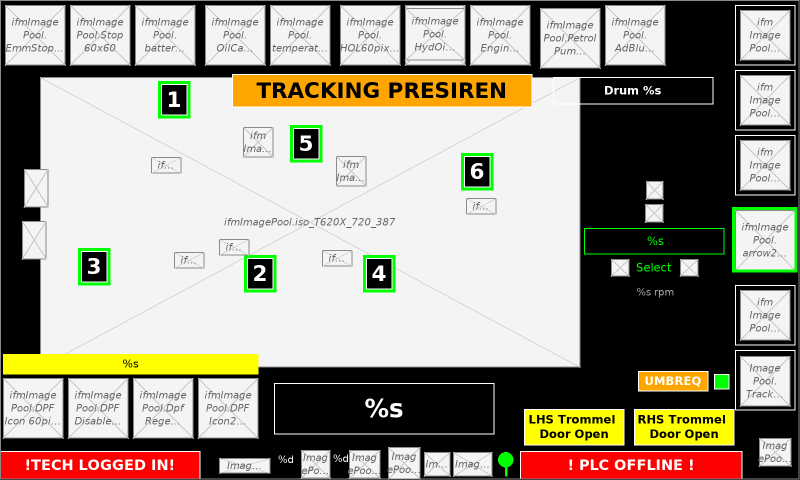
VISUALIZATION Visualization_Main_1  // 800x480
    Frame (0,0 800x480)
        shows Visualization_Main_Status_Common()
    Frame (0,0 800x480)
        shows Visualization_Template()
    Frame (0,0 800x480)
        shows Visualization_Main_Status_Common()
        shows Visualization_Main_Status_Radial()
    Image (740,10 50x50), invisible if: AutoManSelButtons.AutoStartShow=0, image: ifmImagePool.start50pixel
    Image (740,75 50x50), invisible if: AutoManSelButtons.AutoStopShow=0, image: ifmImagePool.Stop Button50pixel
    RoundedRectangle (735,5 60x60)
    RoundedRectangle (735,70 60x60)
    RoundedRectangle (735,135 60x60)
    RoundedRectangle (735,285 60x60)
    RoundedRectangle (735,350 60x60)
    Image (740,140 50x50), image: ifmImagePool.Maintenance50pixel
    RoundedRectangle (735,350 60x60)
    Image (740,290 50x50), image: ifmImagePool.speedometer50pixel
    Image (735,210 60x60), image: ifmImagePool.arrow2_60pixel
    RoundedRectangle (732,207 65x65), invisible if: AutoManSelButtons.Mimic_Halo_RPM_Up_Down=0
        p3450524324: GVL_Viz.SelColor_DWORD
    Image (740,356 50x50), image: ImagePool.Track_50_50
    Rectangle (714,374 15x15), invisible if: GVL_Machine.TrackingModeAllow=0
    RoundedRectangle (524,409 100x36), "LHS Trommel Door Open", invisible if: Machine_IO.Inputs.LHS_TROMMELDOORSW.Dig
    RoundedRectangle (634,409 100x36), "RHS Trommel Door Open", invisible if: Machine_IO.Inputs.RHS_TROMMELDOORSW.Dig
    RoundedRectangle (553,77 160x27), "Drum %s", text variable: GVL_Machine.DrumPressMsg
    RoundedRectangle (638,371 70x20), "UMBREQ", invisible if: Machine_IO.Inputs.UMBTRACKREQ.Dig=0
END_VISUALIZATION

// Device/Application/App_Common/Vizualisations/Main/Visualization_Engine_1
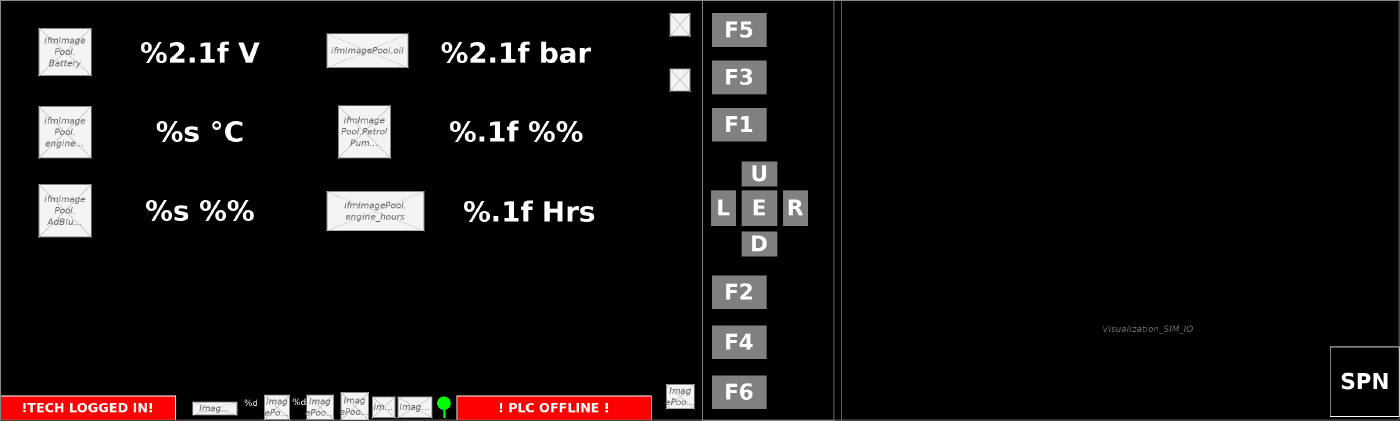
VISUALIZATION Visualization_Engine_1  // 1595x480
    Frame (0,0 800x480)
        shows Visualization_Template()
    Image (385,120 60x60), image: ifmImagePool.Petrol Pump60pixel
    Rectangle (100,20 256x81), "%2.1f V", text variable: GVL_Engine.EngineVoltage
    RoundedRectangle (1515,395 80x80), "SPN"
    Rectangle (460,20 256x81), "%2.1f bar", text variable: GVL_Engine.OilPress_bar/100
    Rectangle (100,110 256x81), "%s °C", text variable: GVL_Engine.CoolantTemperature_degC
    Rectangle (100,200 256x81), "%s %%", text variable: GVL_Engine.Def_TankLevelPercent
    Rectangle (490,201 226x81), "%.1f Hrs", text variable: GVL_Engine.EngineHrs
    Image (385,120 60x60), image: ifmImagePool.Petrol Pump60pixel
    Image (385,120 60x60), invisible if: GVL_Alarms.LowFuelAlarm=0, image: ifmImagePool.Petrol PumpRed60pixel
    Rectangle (460,110 256x81), "%.1f %%", text variable: Machine_IO.Inputs.FUELLEVEL_PERCENT.ScaledReal
    Image (44,210 60x60), image: ifmImagePool.AdBlue Icon On Black60pixel
    Image (372,38 93x39), image: ifmImagePool.oil
    Image (44,121 60x59), image: ifmImagePool.engine_temp
    Image (44,32 60x54), image: ifmImagePool.Battery
    Image (372,218 111x45), image: ifmImagePool.engine_hours
    Image (763,15 23x26), invisible if: Nav.Footer_ShowNavLeft=0, image: ImagePool.Page_nav_left
    Image (763,78 23x26), invisible if: Nav.Footer_ShowNavRight=0, image: ImagePool.Page_nav_right
END_VISUALIZATION

// Device/Application/App_Common/Vizualisations/Main/Visualization_Engine_2
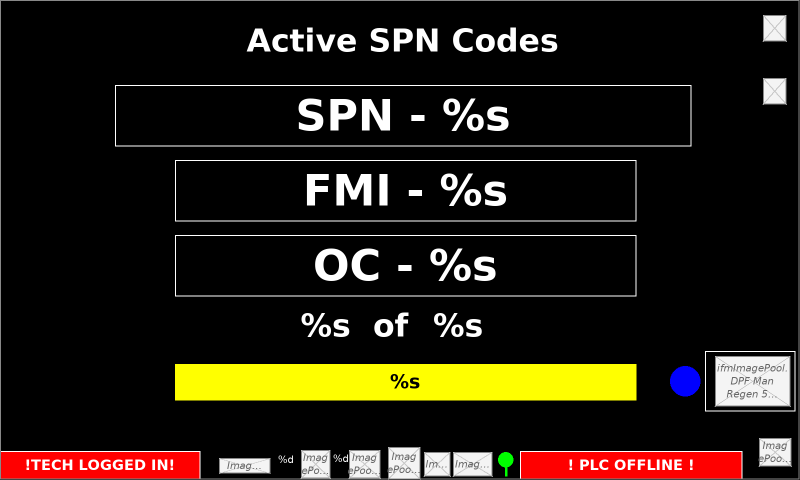
VISUALIZATION Visualization_Engine_2  // 800x480
    Frame (0,0 800x480)
        shows Visualization_Template()
    Rectangle (115,15 576x51), "Active SPN Codes"
    Rectangle (115,85 576x61), "SPN - %s", text variable: GVL_Engine.DM1_Index_SPN
    Rectangle (175,160 461x61), "FMI - %s", text variable: GVL_Engine.DM1_Index_FMI
    Rectangle (175,235 461x61), "OC - %s", text variable: GVL_Engine.DM1_Index_OC
    Rectangle (175,300 236x51), "%s of", text variable: GVL_Engine.DM1_Index
    Rectangle (430,300 206x51), "%s", text variable: GVL_Engine.QtyOf_SPN_Codes
    Image (715,356 75x50), image: ifmImagePool.DPF Man Regen 50 pixelhigh
    Ellipse (670,366 30x30), invisible if: GVL_Engine.ElevateRpmAllowed=FALSE
    RoundedRectangle (705,351 90x60)
    Image (763,15 23x26), invisible if: Nav.Footer_ShowNavLeft=0, image: ImagePool.Page_nav_left
    Image (763,78 23x26), invisible if: Nav.Footer_ShowNavRight=0, image: ImagePool.Page_nav_right
    RoundedRectangle (175,364 461x36), "%s", text variable: GVL_Engine.DPF_Regen_Status_String
END_VISUALIZATION

// Device/Application/App_Common/Vizualisations/Main/Visualization_Settings_2
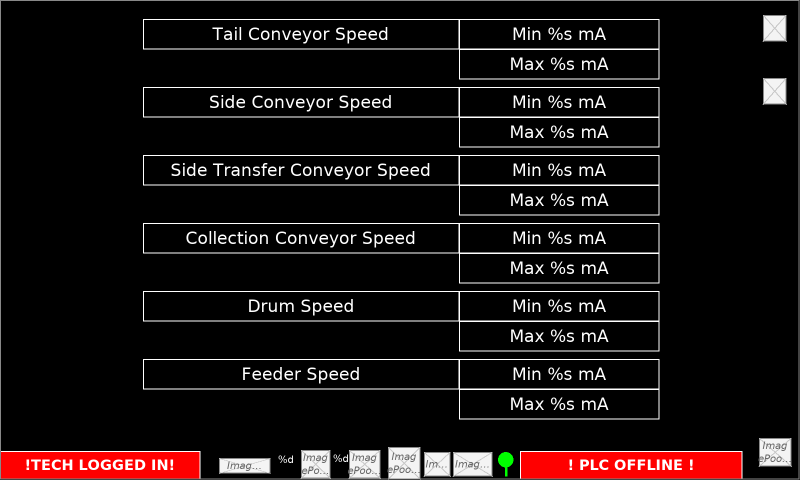
VISUALIZATION Visualization_Settings_2  // 800x480
    Frame (0,0 800x480)
        shows Visualization_Template()
    Rectangle (459,19 200x30), "Min %s mA", text variable: GVL_Persistant.App_Settings.TailConvSpd_Min_mA
        OnMouseClick: write the text variable via VisuDialogs_Template.Numpad, min 0, max GVL_Persistant.App_Settings.TailConvSpd_Max_mA, title "Tail Conveyor Speed Min"
    Rectangle (143,19 316x30), "Tail Conveyor Speed"
    Rectangle (459,49 200x30), "Max %s mA", text variable: GVL_Persistant.App_Settings.TailConvSpd_Max_mA
        OnMouseClick: write the text variable via VisuDialogs_Template.Numpad, min GVL_Persistant.App_Settings.TailConvSpd_Min_mA, max GVL_Persistant.App_Settings.Valve_mA_Max, title "Tail Conveyor Speed Max"
    Rectangle (459,87 200x30), "Min %s mA", text variable: GVL_Persistant.App_Settings.SideConvSpd_Min_mA
        OnMouseClick: write the text variable via VisuDialogs_Template.Numpad, min 0, max GVL_Persistant.App_Settings.SideConvSpd_Max_mA, title "Side Conveyor Speed Min"
    Rectangle (143,87 316x30), "Side Conveyor Speed"
    Rectangle (459,117 200x30), "Max %s mA", text variable: GVL_Persistant.App_Settings.SideConvSpd_Max_mA
        OnMouseClick: write the text variable via VisuDialogs_Template.Numpad, min GVL_Persistant.App_Settings.SideConvSpd_Min_mA, max GVL_Persistant.App_Settings.Valve_mA_Max, title "Side Conveyor Speed Max"
    Rectangle (459,155 200x30), "Min %s mA", text variable: GVL_Persistant.App_Settings.SideTransferConvSpd_Min_mA
        OnMouseClick: write the text variable via VisuDialogs_Template.Numpad, min 0, max GVL_Persistant.App_Settings.SideTransferConvSpd_Max_mA, title "Side Transfer Conveyor Speed Min"
    Rectangle (143,155 316x30), "Side Transfer Conveyor Speed"
    Rectangle (459,185 200x30), "Max %s mA", text variable: GVL_Persistant.App_Settings.SideTransferConvSpd_Max_mA
        OnMouseClick: write the text variable via VisuDialogs_Template.Numpad, min GVL_Persistant.App_Settings.SideTransferConvSpd_Min_mA, max GVL_Persistant.App_Settings.Valve_mA_Max, title "Side Transfer Conveyor Speed Max"
    Rectangle (459,223 200x30), "Min %s mA", text variable: GVL_Persistant.App_Settings.CollectConvSpd_Min_mA
        OnMouseClick: write the text variable via VisuDialogs_Template.Numpad, min 0, max GVL_Persistant.App_Settings.CollectConvSpd_Max_mA, title "Collection Conveyor Speed Min"
    Rectangle (143,223 316x30), "Collection Conveyor Speed"
    Rectangle (459,253 200x30), "Max %s mA", text variable: GVL_Persistant.App_Settings.CollectConvSpd_Max_mA
        OnMouseClick: write the text variable via VisuDialogs_Template.Numpad, min GVL_Persistant.App_Settings.CollectConvSpd_Min_mA, max GVL_Persistant.App_Settings.Valve_mA_Max, title "Collection Conveyor Speed Max"
    Rectangle (459,291 200x30), "Min %s mA", text variable: GVL_Persistant.App_Settings.DrumSpd_Min_mA
        OnMouseClick: write the text variable via VisuDialogs_Template.Numpad, min 0, max GVL_Persistant.App_Settings.DrumSpd_Max_mA, title "Drum Speed Min"
    Rectangle (143,291 316x30), "Drum Speed"
    Rectangle (459,321 200x30), "Max %s mA", text variable: GVL_Persistant.App_Settings.DrumSpd_Max_mA
        OnMouseClick: write the text variable via VisuDialogs_Template.Numpad, min GVL_Persistant.App_Settings.DrumSpd_Min_mA, max GVL_Persistant.App_Settings.Valve_mA_Max, title "Drum Speed Max"
    Rectangle (459,359 200x30), "Min %s mA", text variable: GVL_Persistant.App_Settings.FeederSpd_Min_mA
        OnMouseClick: write the text variable via VisuDialogs_Template.Numpad, min 0, max GVL_Persistant.App_Settings.FeederSpd_Max_mA, title "Feeder Speed Min"
    Rectangle (143,359 316x30), "Feeder Speed"
    Rectangle (459,389 200x30), "Max %s mA", text variable: GVL_Persistant.App_Settings.FeederSpd_Max_mA
        OnMouseClick: write the text variable via VisuDialogs_Template.Numpad, min GVL_Persistant.App_Settings.FeederSpd_Min_mA, max GVL_Persistant.App_Settings.Valve_mA_Max, title "Feeder Speed Max"
    Image (763,15 23x26), invisible if: Nav.Footer_ShowNavLeft=0, image: ImagePool.Page_nav_left
    Image (763,78 23x26), invisible if: Nav.Footer_ShowNavRight=0, image: ImagePool.Page_nav_right
END_VISUALIZATION

// Device/Application/App_Common/Vizualisations/Main/Layout/Visualization_Main_Status_Common
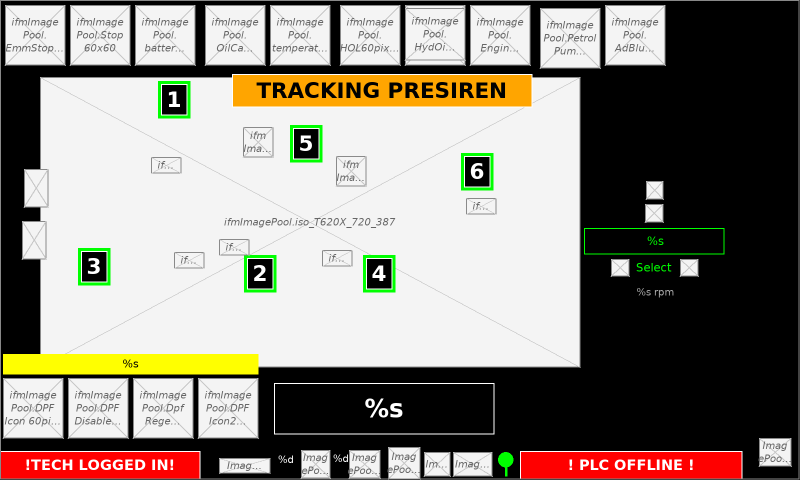
VISUALIZATION Visualization_Main_Status_Common  // 800x480
    Frame (0,0 800x480)
        shows Visualization_Template()
    Frame (0,0 800x480), frame switch variable: TO_INT(GVL_APP.MachineModelRadial)
        shows Visualization_Main_Status_Standard()
        shows Visualization_Main_Status_Radial()
    Image (135,5 60x60), invisible if: GVL_Machine.ChargeLamp=FALSE, image: ifmImagePool.batteryREDonBlack60pixel
    Image (205,5 60x60), invisible if: GVL_Engine.EngineLowOilPressAlarm=FALSE, image: ifmImagePool.OilCanREDonBlack60pixel
    Image (270,5 60x60), invisible if: GVL_Engine.EngineHiTempAlarm=FALSE, image: ifmImagePool.temperatureREDonBlack60pixel
    Image (340,5 60x60), invisible if: GVL_Alarms.LowHydOilAlarm=FALSE, image: ifmImagePool.HOL60pixel
    Image (405,5 60x60), invisible if: GVL_Alarms.HydTempAlarm=FALSE, image: ifmImagePool.HydOilTemp60pixel
    Image (5,5 60x60), invisible if: Safety_Common.ESTOP_HEALHTY_COMMON=0, image: ifmImagePool.EmmStop60pixel
    Image (198,378 60x60), invisible if: GVL_Engine.MILamp=FALSE, image: ifmImagePool.DPF Icon2_60pixel
    Image (133,378 60x60), invisible if: GVL_Engine.DPF_RegenActive=FALSE, image: ifmImagePool.Dpf Regen Active60pixel
    Image (68,378 60x60), invisible if: GVL_Engine.DPF_Regen_Inhibited=FALSE, image: ifmImagePool.DPF Disabled Lamp60pixel
    Image (3,378 60x60), invisible if: GVL_Engine.DPF_Lamp=FALSE, image: ifmImagePool.DPF Icon 60pixel
    Image (70,5 60x60), invisible if: GVL_Machine.UmbMachineShutdown=FALSE, image: ifmImagePool.Stop 60x60
    Image (605,5 60x60), invisible if: GVL_Engine.Def_LowLevLamp=FALSE, image: ifmImagePool.AdBlue Icon On Black60pixel
    Image (470,5 60x60), invisible if: GVL_Engine.EngineWarningLamp=FALSE, image: ifmImagePool.Engine IconAmber60pixel
    Image (470,5 60x60), invisible if: GVL_Engine.DisplayEngineStopLamp=FALSE, image: ifmImagePool.Engine IconRed60pixel
    Image (540,8 60x60), invisible if: PLC_Alarms.Fuel_Symbol_Visible=0, image: ifmImagePool.Petrol PumpRed60pixel
    RoundedRectangle (274,383 220x51), "%s", text variable: GVL_Engine.EngineRpmPerctangeString
    Image (405,8 60x52), invisible if: GVL_Alarms.DrumHighPress_Alarm=0, image: ifmImagePool.HydOil Warning 60 pixel
    RoundedRectangle (232,74 300x33), "TRACKING MODE", invisible if: GVL_Machine.TrackingMode=0
    RoundedRectangle (232,74 300x33), "TRACKING PRESIREN", invisible if: GVL_Machine.TrackPreSiren_Flash=0
    RoundedRectangle (3,354 255x20), "%s", text variable: GVL_Engine.DPF_Regen_Status_String, invisible if: GVL_Engine.DPF_Regen_Status=0
    RoundedRectangle (584,228 140x26), "%s", text variable: AutoManSelButtons.Selected_String, invisible if: LEN(AutoManSelButtons.Selected_String)=0
    Image (646,181 17x18), invisible if: AutoManSelButtons.NavUpShow=0, image: ImagePool.Nav_Up_17_18
    Image (646,204 17x18), invisible if: AutoManSelButtons.NavDownShow=0, image: ImagePool.Nav_Down_17_18
    Image (645,204 18x18), invisible if: AutoManSelButtons.NavCirleShow=0, image: ImagePool.NavCircle_18_18
    Image (611,259 18x17), invisible if: AutoManSelButtons.NavLeftShow=0, image: ImagePool.Nav_Left_17_18
    Image (680,259 18x17), invisible if: AutoManSelButtons.NavRightShow=0, image: ImagePool.Nav_Right_17_18
    RoundedRectangle (629,259 50x17), "Select", text variable: AutoManSelButtons.Selected_String, invisible if: AutoManSelButtons.NavSelectShow=0
    RoundedRectangle (584,279 140x26), "%s rpm", text variable: GVL_Engine.RequestedRPM, invisible if: LEN(AutoManSelButtons.Selected_String)=0
END_VISUALIZATION

// Device/Application/App_Common/Vizualisations/Main/Visualization_Settings_4
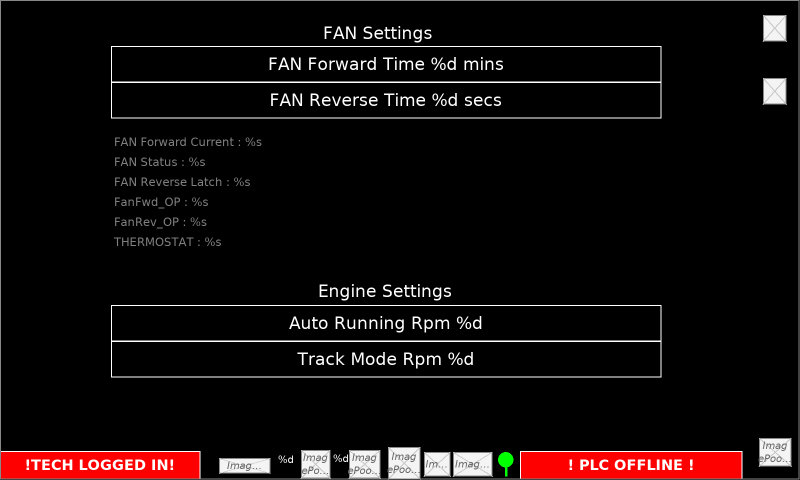
VISUALIZATION Visualization_Settings_4  // 800x480
    Frame (0,0 800x480)
        shows Visualization_Template()
        OnMouseClick: write the text variable via Default, min 0, max 3600, title "Drum Cutout"
    Rectangle (111,46 550x36), "FAN Forward Time %d mins", text variable: GVL_Persistant.App_Settings.Fan_FwdTime_mins
        OnMouseClick: write the text variable via VisuDialogs_Template.Numpad, min 5, max 60, title "FAN Foward Time (mins)"
    Rectangle (155,5 446x56), "FAN Settings"
    Image (763,15 23x26), invisible if: Nav.Footer_ShowNavLeft=0, image: ImagePool.Page_nav_left
    Image (763,78 23x26), invisible if: Nav.Footer_ShowNavRight=0, image: ImagePool.Page_nav_right
    Rectangle (111,82 550x36), "FAN Reverse Time %d secs", text variable: GVL_Persistant.App_Settings.Fan_RevTime_secs
        OnMouseClick: write the text variable via VisuDialogs_Template.Numpad, min 30, max 1200, title "FAN Reverse Time"
    Rectangle (111,132 550x20), "FAN Forward Current : %s", text variable: PLC_FanCtrl.Current_Forward_Time_STR
    Rectangle (111,152 550x20), "FAN Status : %s", text variable: PLC_FanCtrl.STATUS_STRING
    Rectangle (111,172 550x20), "FAN Reverse Latch : %s", text variable: GVL_Persistant.App_Run_Vars.Fan_Reverse_Latch
    Rectangle (111,192 550x20), "FanFwd_OP : %s", text variable: TO_BOOL(Machine_IO.Outputs.FanFwd_OP.Dig)
    Rectangle (111,212 550x20), "FanRev_OP : %s", text variable: TO_BOOL(Machine_IO.Outputs.FanRev_OP.Dig)
    Rectangle (111,232 550x20), "THERMOSTAT : %s", text variable: PLC_FanCtrl.THERMOSTAT
    Rectangle (111,305 550x36), "Auto Running Rpm %d", text variable: GVL_Persistant.App_Settings.AutoRunningRpm
        OnMouseClick: write the text variable via VisuDialogs_Template.Numpad, min GVL_Persistant.App_Settings.AutoRunningRpmMin, max GVL_Persistant.App_Settings.AutoRunningRpmMax, title "Auto Running Rpm"
    Rectangle (162,263 446x56), "Engine Settings"
    Rectangle (111,341 550x36), "Track Mode Rpm %d", text variable: GVL_Persistant.App_Settings.TrackModeRpm
        OnMouseClick: write the text variable via VisuDialogs_Template.Numpad, min GVL_Persistant.App_Settings.TrackModeRpmMin, max GVL_Persistant.App_Settings.TrackModeRpmMax, title "Auto Running Rpm"
END_VISUALIZATION

// /Visualization
VISUALIZATION Visualization  // 1024x768
END_VISUALIZATION

// /Visualization_1
VISUALIZATION Visualization_1  // 1024x768
END_VISUALIZATION

// Device/Application/App_Common/Vizualisations/DIAG_IO/Visualization_DIAG_IO_AUX
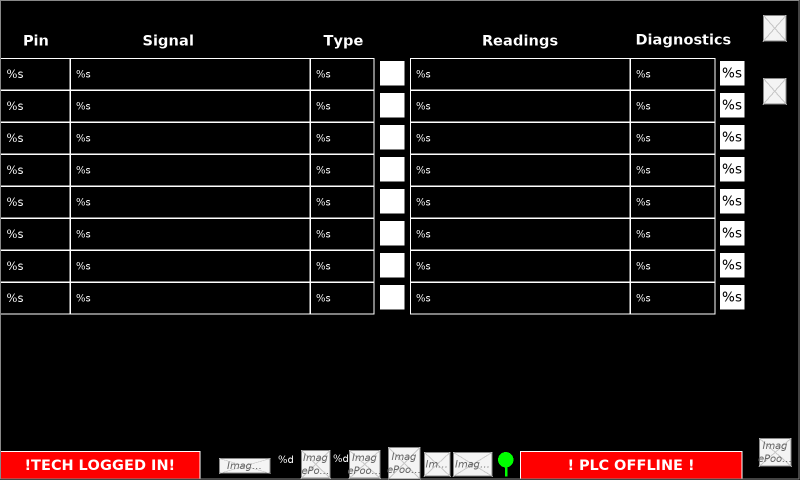
VISUALIZATION Visualization_DIAG_IO_AUX  // 800x480
    Frame (0,0 800x480)
        shows Visualization_Template()
    Image (763,15 23x26), invisible if: Nav.Footer_ShowNavLeft=0, image: ImagePool.Page_nav_left
    Image (763,78 23x26), invisible if: Nav.Footer_ShowNavRight=0, image: ImagePool.Page_nav_right
    Frame (0,25 750x420)
        shows Visualization_CR0403_Op()
END_VISUALIZATION

// Device/Application/App_Common/Vizualisations/DIAG_IO/CR0403/Output_IFM_PLC_CR0403
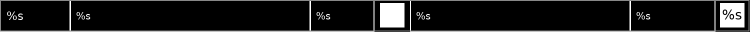
VISUALIZATION Output_IFM_PLC_CR0403  // 750x32
VAR_IN_OUT
	Output: CR0403_Output_Display;
END_VAR
VAR
END_VAR
    Textfield (70,0 240x32), "%s", text variable: Output.oSignalNameStr
    Textfield (0,0 70x32), "%s", text variable: Output.oPinDetailsStr
    Rectangle (380,3 24x24), invisible if: NOT Output.oShowDigRect, colour variable: Output.oDigRectColour
        p3450524324: Output.oDigRectColour
    Textfield (310,0 64x32), "%s", text variable: Output.oTypeStr
    Rectangle (720,3 24x24), "%s", text variable: Output.oForceText, invisible if: NOT HMI_IO.Outputs_EnableAutoMan, input disabled if: NOT HMI_IO.Outputs_EnableAutoMan OR GVL_System.HMI_OP_FORCE_DISABLE, colour variable: Output.oForceColour
        p3450524324: Output.oForceColour
        OnMouseClick:  Dialog=Output_Force, Parameters={flags: , pOutputState: Output.OpREF.OUTPUT_STATE_DATA}, Selected={1: , 0: }, OpenModal=True, OpenCentered=True
    Textfield (630,0 85x32), "%s", text variable: Output.oDiagStr
        p55702900: Output.oMainStringColour
    Textfield (410,0 220x32), "%s", text variable: Output.oMainString
        p55702900: Output.oMainStringColour
END_VISUALIZATION

// Device/Application/App_Common/Vizualisations/DIAG_IO/CR0403/Visualization_CR0403_Op
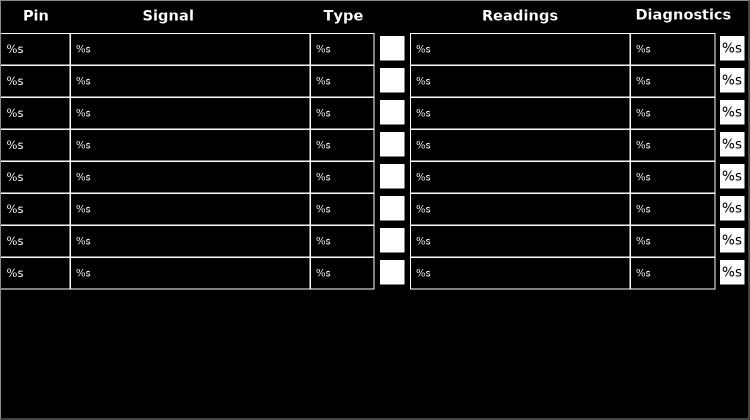
VISUALIZATION Visualization_CR0403_Op  // 750x420
    Frame (0,0 800x32)
        shows Output_IFM_PLC_CRXXXX_TITLE()
    Frame (0,33 750x32)
        shows Output_IFM_PLC_CR0403(Output := HMI_IO.AUX.OP0)
    Frame (0,65 750x32)
        shows Output_IFM_PLC_CR0403(Output := HMI_IO.AUX.OP1)
    Frame (0,97 750x32)
        shows Output_IFM_PLC_CR0403(Output := HMI_IO.AUX.OP2)
    Frame (0,129 750x32)
        shows Output_IFM_PLC_CR0403(Output := HMI_IO.AUX.OP3)
    Frame (0,161 750x32)
        shows Output_IFM_PLC_CR0403(Output := HMI_IO.AUX.OP4)
    Frame (0,193 750x32)
        shows Output_IFM_PLC_CR0403(Output := HMI_IO.AUX.OP5)
    Frame (0,225 750x32)
        shows Output_IFM_PLC_CR0403(Output := HMI_IO.AUX.OP6)
    Frame (0,257 750x32)
        shows Output_IFM_PLC_CR0403(Output := HMI_IO.AUX.OP7)
END_VISUALIZATION

// Device/Application/App_Common/Vizualisations/Main/Layout/Visualization_Main_Status_Radial
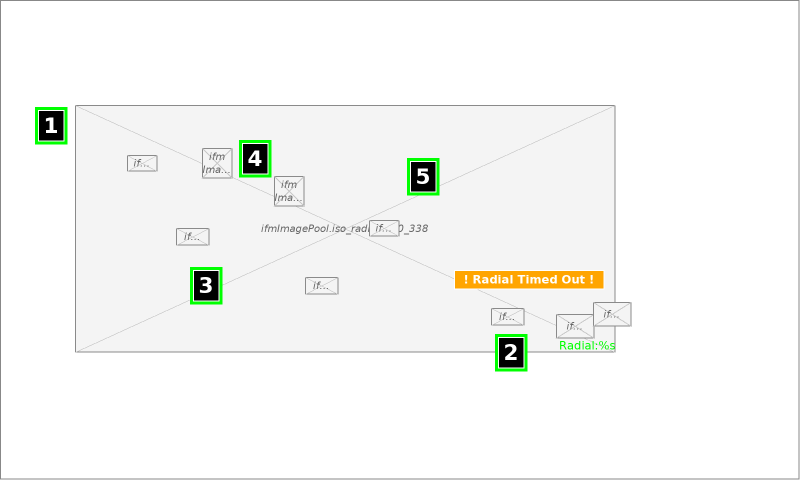
VISUALIZATION Visualization_Main_Status_Radial  // 800x480
    Image (75,105 540x247), image: ifmImagePool.iso_radial_720_338
    Image (369,220 30x16), angle 200, invisible if: Page_Ctrl.Radial_Feeder.Invisible, image: ifmImagePool.Right Arrow Simple 30 pixel wide
        p3560616238: Page_Ctrl.Radial_Feeder.OutX
        p2738717112: Page_Ctrl.Radial_Feeder.OutY
    RoundedRectangle (38,110 26x31), "1", colour variable: AutoManSelButtons.Icon_1_Fill_Colour
    RoundedRectangle (498,337 26x31), "2", colour variable: AutoManSelButtons.Icon_2_Fill_Colour
    RoundedRectangle (410,161 26x31), "5", colour variable: AutoManSelButtons.Icon_5_Fill_Colour
    RoundedRectangle (193,270 26x31), "3", colour variable: AutoManSelButtons.Icon_3_Fill_Colour
    RoundedRectangle (242,143 26x31), "4", colour variable: AutoManSelButtons.Icon_4_Fill_Colour
    Image (274,176 30x30), invisible if: Page_Ctrl.DrumArrow.Invisible, image: ifmImagePool.Rotating Arrow30pixel
        p2858320360: Page_Ctrl.DrumArrow.Out+90
    RoundedRectangle (35,107 32x37), invisible if: AutoManSelButtons.Mimic_Halo_1=0
        p3450524324: GVL_Viz.SelColor_DWORD
    RoundedRectangle (495,334 32x37), invisible if: AutoManSelButtons.Mimic_Halo_2=0
        p3450524324: GVL_Viz.SelColor_DWORD
    RoundedRectangle (239,140 32x37), invisible if: AutoManSelButtons.Mimic_Halo_4=0
        p3450524324: GVL_Viz.SelColor_DWORD
    RoundedRectangle (407,158 32x37), invisible if: AutoManSelButtons.Mimic_Halo_5=0
        p3450524324: GVL_Viz.SelColor_DWORD
    Image (202,148 30x30), invisible if: Page_Ctrl.DrumArrow.Invisible, image: ifmImagePool.Rotating Arrow30pixel
        p2858320360: Page_Ctrl.DrumArrow.Out
    Image (176,228 33x17), angle 22, invisible if: Page_Ctrl.Radial_CollectionArrow_Flat.Invisible, image: ifmImagePool.Right Arrow Simple 30 pixel wide
        p3560616238: Page_Ctrl.Radial_CollectionArrow_Flat.OutX
        p2738717112: Page_Ctrl.Radial_CollectionArrow_Flat.OutY
    Image (491,308 33x17), angle -12, invisible if: Page_Ctrl.Radial_StockpileArrow.Invisible, image: ifmImagePool.Right Arrow Simple 30 pixel wide
        p3560616238: Page_Ctrl.Radial_StockpileArrow.OutX
        p2738717112: Page_Ctrl.Radial_StockpileArrow.OutY
    Image (127,155 30x16), angle 229, invisible if: Page_Ctrl.Radial_TailConveyor.Invisible, image: ifmImagePool.Right Arrow Simple 30 pixel wide
        p3560616238: Page_Ctrl.Radial_TailConveyor.OutX
        p2738717112: Page_Ctrl.Radial_TailConveyor.OutY
    Image (305,277 33x17), angle -1, invisible if: Page_Ctrl.Radial_CollectionArrow_Flat.Invisible, image: ifmImagePool.Right Arrow Simple 30 pixel wide
        p3560616238: Page_Ctrl.Radial_CollectionArrow_Ramp.OutX
        p2738717112: Page_Ctrl.Radial_CollectionArrow_Ramp.OutY
    RoundedRectangle (190,267 32x37), invisible if: AutoManSelButtons.Mimic_Halo_3=0
        p3450524324: GVL_Viz.SelColor_DWORD
    RoundedRectangle (454,270 150x19), "! Radial Timed Out !", invisible if: GVL_APP.RadialTimeOutFlag=0
    Image (556,314 38x24), invisible if: Machine_IO.Outputs.SideConvRaise_RadialLeft_OP.Dig=0, image: ifmImagePool.radial_right
    Image (593,302 38x24), invisible if: Machine_IO.Outputs.SideConvLower_RadialRight_OP.Dig=0, image: ifmImagePool.radial_left
    RoundedRectangle (556,336 150x19), "Radial:%s", text variable: PLC_RadialMode.STATUS_STRING
END_VISUALIZATION

// Device/Application/App_Common/Vizualisations/Main/Layout/Visualization_Main_Status_Standard
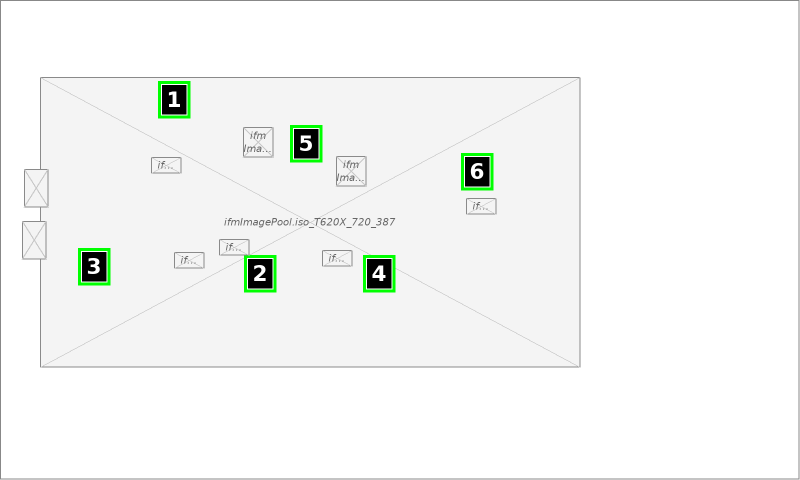
VISUALIZATION Visualization_Main_Status_Standard  // 800x480
    Image (40,77 540x290), image: ifmImagePool.iso_T620X_720_387
    Image (466,198 30x16), angle 198, invisible if: Page_Ctrl.Standard_FeederArrow.Invisible, image: ifmImagePool.Right Arrow Simple 30 pixel wide
        p3560616238: Page_Ctrl.Standard_FeederArrow.OutX
        p2738717112: Page_Ctrl.Standard_FeederArrow.OutY
    RoundedRectangle (161,84 26x31), "1", colour variable: AutoManSelButtons.Icon_1_Fill_Colour
    RoundedRectangle (81,251 26x31), "3", colour variable: AutoManSelButtons.Icon_3_Fill_Colour
    RoundedRectangle (464,156 26x31), "6", colour variable: AutoManSelButtons.Icon_6_Fill_Colour
    RoundedRectangle (293,128 26x31), "5", colour variable: AutoManSelButtons.Icon_5_Fill_Colour
    RoundedRectangle (247,258 26x31), "2", colour variable: AutoManSelButtons.Icon_2_Fill_Colour
    RoundedRectangle (366,258 26x31), "4", colour variable: AutoManSelButtons.Icon_4_Fill_Colour
    Image (322,250 30x16), angle 198, invisible if: Page_Ctrl.Standard_CollectionArrow.Invisible, image: ifmImagePool.Right Arrow Simple 30 pixel wide
        p3560616238: Page_Ctrl.Standard_CollectionArrow.OutX
        p2738717112: Page_Ctrl.Standard_CollectionArrow.OutY
    Image (243,127 30x30), invisible if: Page_Ctrl.DrumArrow.Invisible, image: ifmImagePool.Rotating Arrow30pixel
        p2858320360: Page_Ctrl.DrumArrow.Out
    RoundedRectangle (158,81 32x37), invisible if: AutoManSelButtons.Mimic_Halo_1=0
        p3450524324: GVL_Viz.SelColor_DWORD
    RoundedRectangle (244,255 32x37), invisible if: AutoManSelButtons.Mimic_Halo_2=0
        p3450524324: GVL_Viz.SelColor_DWORD
    RoundedRectangle (78,248 32x37), invisible if: AutoManSelButtons.Mimic_Halo_3=0
        p3450524324: GVL_Viz.SelColor_DWORD
    RoundedRectangle (363,255 32x37), invisible if: AutoManSelButtons.Mimic_Halo_4=0
        p3450524324: GVL_Viz.SelColor_DWORD
    RoundedRectangle (290,125 32x37), invisible if: AutoManSelButtons.Mimic_Halo_5=0
        p3450524324: GVL_Viz.SelColor_DWORD
    RoundedRectangle (461,153 32x37), invisible if: AutoManSelButtons.Mimic_Halo_6=0
        p3450524324: GVL_Viz.SelColor_DWORD
    Image (336,156 30x30), invisible if: Page_Ctrl.DrumArrow.Invisible, image: ifmImagePool.Rotating Arrow30pixel
        p2858320360: Page_Ctrl.DrumArrow.Out+90
    Image (174,252 30x16), angle 198, invisible if: Page_Ctrl.Standard_SideConvArrow.Invisible, image: ifmImagePool.Right Arrow Simple 30 pixel wide
        p3560616238: Page_Ctrl.Standard_SideConvArrow.OutX
        p2738717112: Page_Ctrl.Standard_SideConvArrow.OutY
    Image (219,239 30x16), angle 161, invisible if: Page_Ctrl.Standard_SideTransferArrow.Invisible, image: ifmImagePool.Right Arrow Simple 30 pixel wide
        p3560616238: Page_Ctrl.Standard_SideTransferArrow.OutX
        p2738717112: Page_Ctrl.Standard_SideTransferArrow.OutY
    Image (151,157 30x16), angle 224, invisible if: Page_Ctrl.Standard_TailConvArrow.Invisible, image: ifmImagePool.Right Arrow Simple 30 pixel wide
        p3560616238: Page_Ctrl.Standard_TailConvArrow.OutX
        p2738717112: Page_Ctrl.Standard_TailConvArrow.OutY
    Image (24,169 24x38), invisible if: Machine_IO.Outputs.SideConvRaise_RadialLeft_OP.Dig=0, image: ifmImagePool.side_conv_up
    Image (22,221 24x38), invisible if: Machine_IO.Outputs.SideConvLower_RadialRight_OP.Dig=0, image: ifmImagePool.side_conv_down
END_VISUALIZATION

// Device/Application/App_Common/Vizualisations/Main/Visualization_Settings_3
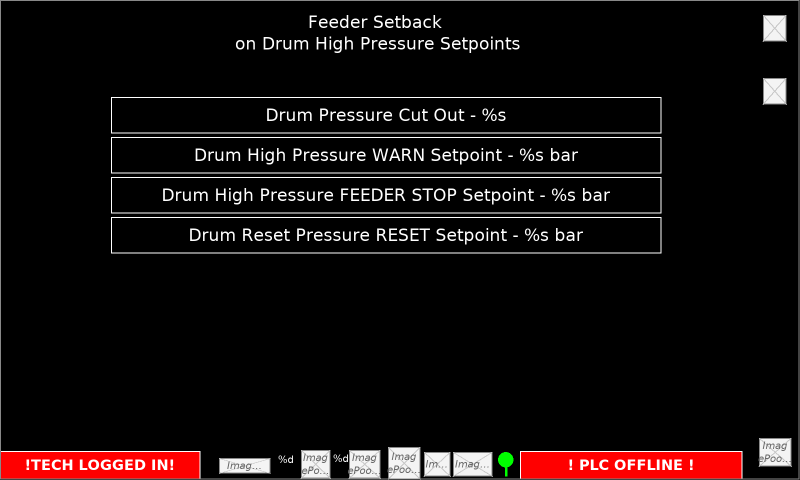
VISUALIZATION Visualization_Settings_3  // 800x480
    Frame (0,0 800x480)
        shows Visualization_Template()
        OnMouseClick: write the text variable via Default, min 0, max 3600, title "Drum Cutout"
    Rectangle (111,97 550x36), "Drum Pressure Cut Out - %s", text variable: GVL_Persistant.App_Settings.EnableDrumPressCutOut
        toggle GVL_Persistant.App_Settings.EnableDrumPressCutOut
    Rectangle (111,137 550x36), "Drum High Pressure WARN Setpoint - %s bar", text variable: GVL_Persistant.App_Settings.DrumPressHi_SP
        OnMouseClick: write the text variable via VisuDialogs_Template.Numpad, min GVL_Persistant.App_Settings.DrumPressReset_SP, max GVL_Persistant.App_Settings.DrumPressHiHi_SP, title "Drum High Press Warn SP"
    Rectangle (111,177 550x36), "Drum High Pressure FEEDER STOP Setpoint - %s bar", text variable: GVL_Persistant.App_Settings.DrumPressHiHi_SP
        OnMouseClick: write the text variable via VisuDialogs_Template.Numpad, min GVL_Persistant.App_Settings.DrumPressHi_SP, max GVL_Persistant.App_Settings.DrumPressMax
    Rectangle (111,217 550x36), "Drum Reset Pressure RESET Setpoint - %s bar", text variable: GVL_Persistant.App_Settings.DrumPressReset_SP
        OnMouseClick: write the text variable via VisuDialogs_Template.Numpad, min 0, max GVL_Persistant.App_Settings.DrumPressHi_SP
    Rectangle (155,5 446x56), "Feeder Setback on Drum High Pressure Setpoints"
    Image (763,15 23x26), invisible if: Nav.Footer_ShowNavLeft=0, image: ImagePool.Page_nav_left
    Image (763,78 23x26), invisible if: Nav.Footer_ShowNavRight=0, image: ImagePool.Page_nav_right
END_VISUALIZATION

// Device/Application/App_Common/Vizualisations/Main/Visualization_Engine_3
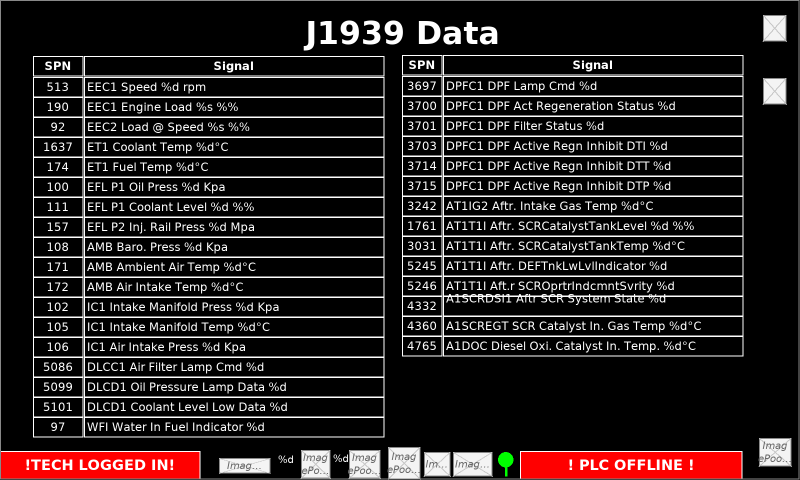
VISUALIZATION Visualization_Engine_3  // 800x480
    Frame (0,0 800x480)
        shows Visualization_Template()
    Image (763,15 23x26), invisible if: Nav.Footer_ShowNavLeft=0, image: ImagePool.Page_nav_left
    Image (763,78 23x26), invisible if: Nav.Footer_ShowNavRight=0, image: ImagePool.Page_nav_right
    Rectangle (84,77 300x20), "EEC1 Speed %d rpm", text variable: TO_INT(GVL_J1939.EEC1_EngSpeed)
    Rectangle (84,97 300x20), "EEC1 Engine Load %s %%", text variable: GVL_J1939.EEC1_ActualEngPercentTorque
    Rectangle (84,117 300x20), "EEC2 Load @ Speed %s %%", text variable: GVL_J1939.EEC2_EngPercentLoadAtCurrentSpeed
    Rectangle (84,137 300x20), "ET1 Coolant Temp %d°C", text variable: TO_INT(GVL_J1939.ET1_EngCoolantTemp)
    Rectangle (84,157 300x20), "ET1 Fuel Temp %d°C", text variable: TO_INT(GVL_J1939.ET1_EngFuelTemp1)
    Rectangle (84,197 300x20), "EFL P1 Coolant Level %d %%", text variable: TO_INT(GVL_J1939.EFL_P1_EngCoolantLevel)
    Rectangle (84,177 300x20), "EFL P1 Oil Press %d Kpa", text variable: TO_INT(GVL_J1939.EFL_P1_EngOilPress)
    Rectangle (84,217 300x20), "EFL P2 Inj. Rail Press %d Mpa", text variable: TO_INT(GVL_J1939.EFL_P2_EngInjectorMeteringRail1Press)
    Rectangle (84,237 300x20), "AMB Baro. Press %d Kpa", text variable: TO_INT(GVL_J1939.AMB_BarometricPress)
    Rectangle (84,257 300x20), "AMB Ambient Air Temp %d°C", text variable: TO_INT(GVL_J1939.AMB_AmbientAirTemp)
    Rectangle (84,277 300x20), "AMB Air Intake Temp %d°C", text variable: TO_INT(GVL_J1939.AMB_EngAirIntakeTemp)
    Rectangle (84,297 300x20), "IC1 Intake Manifold Press %d Kpa", text variable: TO_INT(GVL_J1939.IC1_EngIntakeManifold1Press)
    Rectangle (84,317 300x20), "IC1 Intake Manifold Temp %d°C", text variable: TO_INT(GVL_J1939.IC1_EngIntakeManifold1Temp)
    Rectangle (84,337 300x20), "IC1 Air Intake Press %d Kpa", text variable: TO_INT(GVL_J1939.IC1_EngAirIntakePress)
    Rectangle (84,357 300x20), "DLCC1 Air Filter Lamp Cmd %d", text variable: GVL_J1939.DLCC1_EngAirFilterRestrictionLampCmd
    Rectangle (84,377 300x20), "DLCD1 Oil Pressure Lamp Data %d", text variable: GVL_J1939.DLCD1_EngOilPressLowLampData
    Rectangle (84,397 300x20), "DLCD1 Coolant Level Low Data %d", text variable: GVL_J1939.DLCD1_EngCoolantLevelLowLampData
    Rectangle (84,417 300x20), "WFI Water In Fuel Indicator %d", text variable: GVL_J1939.WFI_WaterInFuelIndicator
    Rectangle (443,76 300x20), "DPFC1 DPF Lamp Cmd %d", text variable: GVL_J1939.DPFC1_DieselParticulateFilterLampCmd
    Rectangle (443,96 300x20), "DPFC1 DPF Act Regeneration Status %d", text variable: GVL_J1939.DPFC1_DslPrtcltFltrActvRgnrtionStatus
    Rectangle (443,116 300x20), "DPFC1 DPF Filter Status %d", text variable: GVL_J1939.DPFC1_DieselParticulateFilterStatus
    Rectangle (443,136 300x20), "DPFC1 DPF Active Regn Inhibit DTI %d", text variable: GVL_J1939.DPFC1_DslPrtcltFltrActvRgnrtnInhbtdDTI
    Rectangle (443,156 300x20), "DPFC1 DPF Active Regn Inhibit DTT %d", text variable: GVL_J1939.DPFC1_DslPrtcltFltrActvRgnrtnInhbtdDTT
    Rectangle (443,176 300x20), "DPFC1 DPF Active Regn Inhibit DTP %d", text variable: GVL_J1939.DPFC1_DslPrtcltFltrActvRgnrtnInhbtdDTP
    Rectangle (402,76 40x20), "3697"
    Rectangle (402,96 40x20), "3700"
    Rectangle (402,116 40x20), "3701"
    Rectangle (402,136 40x20), "3703"
    Rectangle (402,156 40x20), "3714"
    Rectangle (402,176 40x20), "3715"
    Rectangle (33,77 50x20), "513"
    Rectangle (33,97 50x20), "190"
    Rectangle (33,117 50x20), "92"
    Rectangle (33,137 50x20), "1637"
    Rectangle (33,157 50x20), "174"
    Rectangle (33,177 50x20), "100"
    Rectangle (33,197 50x20), "111"
    Rectangle (33,217 50x20), "157"
    Rectangle (33,237 50x20), "108"
    Rectangle (33,257 50x20), "171"
    Rectangle (33,277 50x20), "172"
    Rectangle (33,297 50x20), "102"
    Rectangle (33,317 50x20), "105"
    Rectangle (33,337 50x20), "106"
    Rectangle (33,357 50x20), "5086"
    Rectangle (33,377 50x20), "5099"
    Rectangle (33,397 50x20), "5101"
    Rectangle (33,417 50x20), "97"
    Rectangle (443,196 300x20), "AT1IG2 Aftr. Intake Gas Temp %d°C", text variable: GVL_J1939.AT1IG2_Aftrtrtmnt1DslPrtcltFltrInt_0000
    Rectangle (402,196 40x20), "3242"
    Rectangle (443,216 300x20), "AT1T1I Aftr. SCRCatalystTankLevel %d %%", text variable: GVL_J1939.AT1T1I_Aftrtrtmnt1SCRCatalystTankLevel
    Rectangle (402,216 40x20), "1761"
    Rectangle (443,236 300x20), "AT1T1I Aftr. SCRCatalystTankTemp %d°C", text variable: GVL_J1939.AT1T1I_Aftrtrtment1SCRCatalystTankTemp
    Rectangle (402,236 40x20), "3031"
    Rectangle (443,256 300x20), "AT1T1I Aftr. DEFTnkLwLvlIndicator %d", text variable: GVL_J1939.AT1T1I_Aftrtrtmnt1DEFTnkLwLvlIndicator
    Rectangle (402,256 40x20), "5245"
    Rectangle (443,276 300x20), "AT1T1I Aft.r SCROprtrIndcmntSvrity %d", text variable: GVL_J1939.AT1T1I_AftrtrtmntSCROprtrIndcmntSvrity
    Rectangle (402,276 40x20), "5246"
    Rectangle (443,296 300x20), "A1SCRDSI1 Aftr SCR System State %d", text variable: GVL_J1939.A1SCRDSI1_Aftertreatment1SCRSystemState
    Rectangle (402,296 40x20), "4332"
    Rectangle (443,316 300x20), "A1SCREGT SCR Catalyst In. Gas Temp %d°C", text variable: GVL_J1939.A1SCREGT_Aftrtrtmnt1SCRCtlystIntkGasTemp
    Rectangle (402,316 40x20), "4360"
    Rectangle (443,336 300x20), "A1DOC Diesel Oxi. Catalyst In. Temp. %d°C", text variable: GVL_J1939.A1DOC_Aftrtrtmnt1DslOxdtnCtlystIn_0000
    Rectangle (402,336 40x20), "4765"
    Rectangle (33,56 50x20), "SPN"
    Rectangle (84,56 300x20), "Signal"
    Rectangle (402,55 40x20), "SPN"
    Rectangle (443,55 300x20), "Signal"
    Rectangle (115,15 576x36), "J1939 Data"
END_VISUALIZATION

(* text list System (id | default | ge | en)
  Apr | Apr | Apr | Apr
  April | April | April | April
  Aug | Aug | Aug | Aug
  August | August | August | August
  Dec | Dec | Dec | Dec
  December | December | December | December
  Feb | Feb | Feb | Feb
  February | February | February | February
  Fri | Fri | Fri | Fri
  Friday | Friday | Friday | Friday
  Jan | Jan | Jan | Jan
  January | January | January | January
  Jul | Jul | Jul | Jul
  July | July | July | July
  Jun | Jun | Jun | Jun
  June | June | June | June
  Mar | Mar | Mar | Mar
  March | March | March | March
  May | May | May | May
  May_3Letter | May | May | May
  Mon | Mon | Mon | Mon
  Monday | Monday | Monday | Monday
  Nov | Nov | Nov | Nov
  November | November | November | November
  Oct | Oct | Oct | Oct
  October | October | October | October
  Sat | Sat | Sat | Sat
  Saturday | Saturday | Saturday | Saturday
  Sep | Sep | Sep | Sep
  September | September | September | September
  Sun | Sun | Sun | Sun
  Sunday | Sunday | Sunday | Sunday
  Thu | Thu | Thu | Thu
  Thursday | Thursday | Thursday | Thursday
  Tue | Tue | Tue | Tue
  Tuesday | Tuesday | Tuesday | Tuesday
  Wed | Wed | Wed | Wed
  Wednesday | Wednesday | Wednesday | Wednesday
   |  |  |  *)

(* text list AlarmGroup_IO (id | default | ge | en)
   |  |  |  *)

(* text list AlarmGroup_App (id | default | ge | en)
  101 | Emergencey Stop Active | Emergencey Stop Active | Emergencey Stop Active
  102 | PLC Ethernet Common Failure | PLC Ethernet Common Failure | PLC Ethernet Common Failure
  1100 | Ethernet - CHASSIS PLC Missing on powerup | Ethernet - CHASSIS PLC Missing on powerup | Ethernet - CHASSIS PLC Missing on powerup
  1101 | Ethernet - CHASSIS PLC - heartbeat less than error | Ethernet - CHASSIS PLC - heartbeat less than error | Ethernet - CHASSIS PLC - heartbeat less than error
  1102 | Ethernet - CHASSIS PLC - heartbeat difference error | Ethernet - CHASSIS PLC - heartbeat difference error | Ethernet - CHASSIS PLC - heartbeat difference error
  1103 | Ethernet - CHASSIS PLC - heartbeat frozen error | Ethernet - CHASSIS PLC - heartbeat frozen error | Ethernet - CHASSIS PLC - heartbeat frozen error
  1104 | Ethernet - CHASSIS PLC - heartbeat difference warning | Ethernet - CHASSIS PLC - heartbeat difference warning | Ethernet - CHASSIS PLC - heartbeat difference warning
  1105 | Ethernet - CHASSIS PLC - heartbeat frozen warning | Ethernet - CHASSIS PLC - heartbeat frozen warning | Ethernet - CHASSIS PLC - heartbeat frozen warning
  103 | Battery Voltage Warning | Battery Voltage Warning | Battery Voltage Warning
  104 | Hydraulic Oil level Low Alarm | Hydraulic Oil level Low Alarm | Hydraulic Oil level Low Alarm
  105 | Hydraulic Oil Temperature Alarm | Hydraulic Oil Temperature Alarm | Hydraulic Oil Temperature Alarm
  106 | Drum High Pressure Alarm | Drum High Pressure Alarm | Drum High Pressure Alarm
  107 | Low Fuel Level Alarm | Low Fuel Level Alarm | Low Fuel Level Alarm
  108 | Auto Shutdown Alarm | Auto Shutdown Alarm | Auto Shutdown Alarm
  109 | Engine Low Oil Pressure Alarm | Engine Low Oil Pressure Alarm | Engine Low Oil Pressure Alarm
  110 | Engine High Temperature Alarm | Engine High Temperature Alarm | Engine High Temperature Alarm
   |  |  |  *)

(* text list TextList_IFM_Diag_Codes (id | default | ge | en)
  0 | STAT_INACTIVE | STAT_INACTIVE | STAT_INACTIVE
  1 | STAT_DONE | STAT_DONE | STAT_DONE
  2 | STAT_BUSY | STAT_BUSY | STAT_BUSY
  3 | STAT_PREPARING | STAT_PREPARING | STAT_PREPARING
  4 | STAT_READY | STAT_READY | STAT_READY
  5 | STAT_RESET | STAT_RESET | STAT_RESET
  6 | STAT_ABORTED | STAT_ABORTED | STAT_ABORTED
  7 | RESERVED_07 | RESERVED_07 | RESERVED_07
  8 | RESERVED_08 | RESERVED_08 | RESERVED_08
  9 | RESERVED_09 | RESERVED_09 | RESERVED_09
  10 | ERR_OPEN_CIRCUIT | ERR_OPEN_CIRCUIT | ERR_OPEN_CIRCUIT
  11 | ERR_SHORT_CIRCUIT | ERR_SHORT_CIRCUIT | ERR_SHORT_CIRCUIT
  12 | ERR_OVERLOAD_CURRENT | ERR_OVERLOAD_CURRENT | ERR_OVERLOAD_CURRENT
  13 | ERR_LOW_CURRENT | ERR_LOW_CURRENT | ERR_LOW_CURRENT
  14 | ERR_UNDERVOLTAGE_VBBX | ERR_UNDERVOLTAGE_VBBX | ERR_UNDERVOLTAGE_VBBX
  15 | ERR_OVERVOLTAGE_VBBX | ERR_OVERVOLTAGE_VBBX | ERR_OVERVOLTAGE_VBBX
  16 | ERR_STUCK_AT_HIGH | ERR_STUCK_AT_HIGH | ERR_STUCK_AT_HIGH
  17 | ERR_STUCK_AT_LOW | ERR_STUCK_AT_LOW | ERR_STUCK_AT_LOW
  18 | ERR_HIGH_TEMPERATURE | ERR_HIGH_TEMPERATURE | ERR_HIGH_TEMPERATURE
  19 | ERR_LOW_TEMPERATURE | ERR_LOW_TEMPERATURE | ERR_LOW_TEMPERATURE
  20 | ERR_INVALID_VALUE | ERR_INVALID_VALUE | ERR_INVALID_VALUE
  21 | ERR_INVALID_CHANNEL | ERR_INVALID_CHANNEL | ERR_INVALID_CHANNEL
  22 | ERR_INVALID_MODE | ERR_INVALID_MODE | ERR_INVALID_MODE
  23 | ERR_INVALID_FREQUENCY | ERR_INVALID_FREQUENCY | ERR_INVALID_FREQUENCY
  24 | ERR_INVALID_DITHER | ERR_INVALID_DITHER | ERR_INVALID_DITHER
  25 | ERR_INVALID_FILTER | ERR_INVALID_FILTER | ERR_INVALID_FILTER
  26 | ERR_UNREACHABLE_CURRENT | ERR_UNREACHABLE_CURRENT | ERR_UNREACHABLE_CURRENT
  27 | ERR_SLOW_SIGNAL | ERR_SLOW_SIGNAL | ERR_SLOW_SIGNAL
  28 | ERR_CHANGEOVER_TIME | ERR_CHANGEOVER_TIME | ERR_CHANGEOVER_TIME
  29 | ERR_INSTANCE | ERR_INSTANCE | ERR_INSTANCE
  30 | ERR_INSTANCE_LIMIT | ERR_INSTANCE_LIMIT | ERR_INSTANCE_LIMIT
  31 | ERR_INVALID_COLOUR | ERR_INVALID_COLOUR | ERR_INVALID_COLOUR
  32 | ERR_NO_IDENTITY | ERR_NO_IDENTITY | ERR_NO_IDENTITY
  33 | ERR_ACCESS | ERR_ACCESS | ERR_ACCESS
  34 | ERR_UNDEFINED | ERR_UNDEFINED | ERR_UNDEFINED
  35 | ERR_FUNC_KEY_MISSED | ERR_FUNC_KEY_MISSED | ERR_FUNC_KEY_MISSED
  36 | ERR_BUFFER_OVERFLOW | ERR_BUFFER_OVERFLOW | ERR_BUFFER_OVERFLOW
  37 | ERR_BAUDRATE_ALREADY_SET | ERR_BAUDRATE_ALREADY_SET | ERR_BAUDRATE_ALREADY_SET
  38 | ERR_INACTIVE_INTERFACE | ERR_INACTIVE_INTERFACE | ERR_INACTIVE_INTERFACE
  39 | ERR_TIMEOUT | ERR_TIMEOUT | ERR_TIMEOUT
  40 | ERR_OUT_OF_MEMORY | ERR_OUT_OF_MEMORY | ERR_OUT_OF_MEMORY
  41 | ERR_BUS_OFF | ERR_BUS_OFF | ERR_BUS_OFF
  42 | ERR_BAD_CRC | ERR_BAD_CRC | ERR_BAD_CRC
  43 | ERR_EXCEEDED_RANGE | ERR_EXCEEDED_RANGE | ERR_EXCEEDED_RANGE
  44 | ERR_INTERNAL_COMMUNICATION | ERR_INTERNAL_COMMUNICATION | ERR_INTERNAL_COMMUNICATION
  45 | ERR_NOT_SUPPORTED | ERR_NOT_SUPPORTED | ERR_NOT_SUPPORTED
  46 | ERR_TIMING | ERR_TIMING | ERR_TIMING
  47 | ERR_INTERNAL | ERR_INTERNAL | ERR_INTERNAL
  48 | ERR_FILE_SYSTEM | ERR_FILE_SYSTEM | ERR_FILE_SYSTEM
  49 | ERR_INVALID_IP_CFG | ERR_INVALID_IP_CFG | ERR_INVALID_IP_CFG
  50 | ERR_FAILED_ERR_RESET | ERR_FAILED_ERR_RESET | ERR_FAILED_ERR_RESET
  51 | ERR_DEVICE_NOT_AVAILABLE | ERR_DEVICE_NOT_AVAILABLE | ERR_DEVICE_NOT_AVAILABLE
  52 | ERR_NO_OBJECT | ERR_NO_OBJECT | ERR_NO_OBJECT
  53 | ERR_UNREACHABLE_VOLTAGE | ERR_UNREACHABLE_VOLTAGE | ERR_UNREACHABLE_VOLTAGE
  54 | ERR_AT_GROUP_OUTPUT | ERR_AT_GROUP_OUTPUT | ERR_AT_GROUP_OUTPUT
  55 | ERR_CONTROL_DITHER | ERR_CONTROL_DITHER | ERR_CONTROL_DITHER
  56 | ERR_UNDERVOLTAGE_VBBX_WARNING | ERR_UNDERVOLTAGE_VBBX_WARNING | ERR_UNDERVOLTAGE_VBBX_WARNING
  57 | ERR_OVERVOLTAGE_VBBX_WARNING | ERR_OVERVOLTAGE_VBBX_WARNING | ERR_OVERVOLTAGE_VBBX_WARNING
  58 | ERR_LOW_TEMPERATURE_WARNING | ERR_LOW_TEMPERATURE_WARNING | ERR_LOW_TEMPERATURE_WARNING
  59 | ERR_HIGH_TEMPERATURE_WARNING | ERR_HIGH_TEMPERATURE_WARNING | ERR_HIGH_TEMPERATURE_WARNING
  60 | ERR_RANGE_OVERRUN | ERR_RANGE_OVERRUN | ERR_RANGE_OVERRUN
  61 | ERR_RANGE_UNDERRUN | ERR_RANGE_UNDERRUN | ERR_RANGE_UNDERRUN
  62 | DIAG_INVALID_VALUE | DIAG_INVALID_VALUE | DIAG_INVALID_VALUE
  63 | DIAG_INTERNAL | DIAG_INTERNAL | DIAG_INTERNAL
  64 | DIAG_OPEN_CIRCUIT | DIAG_OPEN_CIRCUIT | DIAG_OPEN_CIRCUIT
  65 | DIAG_SHORT_CIRCUIT | DIAG_SHORT_CIRCUIT | DIAG_SHORT_CIRCUIT
  66 | DIAG_UNDERVOLTAGE_VBBX | DIAG_UNDERVOLTAGE_VBBX | DIAG_UNDERVOLTAGE_VBBX
  67 | DIAG_OVERVOLTAGE_VBBX | DIAG_OVERVOLTAGE_VBBX | DIAG_OVERVOLTAGE_VBBX
  68 | DIAG_OVERLOAD_CURRENT | DIAG_OVERLOAD_CURRENT | DIAG_OVERLOAD_CURRENT
  69 | DIAG_STUCK_AT | DIAG_STUCK_AT | DIAG_STUCK_AT
  70 | DIAG_STUCK_AT_HIGH | DIAG_STUCK_AT_HIGH | DIAG_STUCK_AT_HIGH
  71 | DIAG_STUCK_AT_LOW | DIAG_STUCK_AT_LOW | DIAG_STUCK_AT_LOW
  72 | DIAG_INVALID_COLOUR | DIAG_INVALID_COLOUR | DIAG_INVALID_COLOUR
  73 | DIAG_OVERVOLTAGE | DIAG_OVERVOLTAGE | DIAG_OVERVOLTAGE
  74 | DIAG_UNDERVOLTAGE | DIAG_UNDERVOLTAGE | DIAG_UNDERVOLTAGE
  75 | DIAG_NO_CALIB | DIAG_NO_CALIB | DIAG_NO_CALIB
  76 | DIAG_ACCESS | DIAG_ACCESS | DIAG_ACCESS
  77 | DIAG_CHANGEOVER_TIME | DIAG_CHANGEOVER_TIME | DIAG_CHANGEOVER_TIME
  78 | ERR_OVERVOLTAGE | ERR_OVERVOLTAGE | ERR_OVERVOLTAGE
  79 | ERR_UNDERVOLTAGE | ERR_UNDERVOLTAGE | ERR_UNDERVOLTAGE
  80 | ERR_STUCK_AT | ERR_STUCK_AT | ERR_STUCK_AT
  81 | DIAG_CONTROL_DITHER | DIAG_CONTROL_DITHER | DIAG_CONTROL_DITHER
  82 | DIAG_SLOW_SIGNAL | DIAG_SLOW_SIGNAL | DIAG_SLOW_SIGNAL
  83 | DIAG_DIAG_PRO_MODE | DIAG_DIAG_PRO_MODE | DIAG_DIAG_PRO_MODE
  84 | DIAG_WINDOW | DIAG_WINDOW | DIAG_WINDOW
  85 | ERR_SDO_IDX_NOT_EXIST | ERR_SDO_IDX_NOT_EXIST | ERR_SDO_IDX_NOT_EXIST
  86 | ERR_SDO_SUBIDX_NOT_EXIST | ERR_SDO_SUBIDX_NOT_EXIST | ERR_SDO_SUBIDX_NOT_EXIST
  87 | ERR_SDO_UNSUPPORTED_ACCESS | ERR_SDO_UNSUPPORTED_ACCESS | ERR_SDO_UNSUPPORTED_ACCESS
  88 | ERR_SDO_DATA_TYPE | ERR_SDO_DATA_TYPE | ERR_SDO_DATA_TYPE
  89 | DIAG_LOW_TEMPERATURE | DIAG_LOW_TEMPERATURE | DIAG_LOW_TEMPERATURE
  90 | DIAG_HIGH_TEMPERATURE | DIAG_HIGH_TEMPERATURE | DIAG_HIGH_TEMPERATURE
  91 | DIAG_INVALID_DITHER | DIAG_INVALID_DITHER | DIAG_INVALID_DITHER
  92 | DIAG_INVALID_FREQUENCY | DIAG_INVALID_FREQUENCY | DIAG_INVALID_FREQUENCY
  93 | DIAG_RANGE_OVERRUN | DIAG_RANGE_OVERRUN | DIAG_RANGE_OVERRUN
  94 | DIAG_RANGE_UNDERRUN | DIAG_RANGE_UNDERRUN | DIAG_RANGE_UNDERRUN
  95 | DIAG_INVALID_FILTER | DIAG_INVALID_FILTER | DIAG_INVALID_FILTER
  96 | ERR_COMPARE_MISMATCH | ERR_COMPARE_MISMATCH | ERR_COMPARE_MISMATCH
  97 | DIAG_INVALID_IP_CFG | DIAG_INVALID_IP_CFG | DIAG_INVALID_IP_CFG
  98 | DIAG_LOW_CURRENT | DIAG_LOW_CURRENT | DIAG_LOW_CURRENT
  99 | DIAG_AT_GROUP_OUTPUT | DIAG_AT_GROUP_OUTPUT | DIAG_AT_GROUP_OUTPUT
  100 | ERR_SDO_UNKNOWN | ERR_SDO_UNKNOWN | ERR_SDO_UNKNOWN
  101 | ERR_BAUDRATE_INVALID_OR_ALREADY_SET | ERR_BAUDRATE_INVALID_OR_ALREADY_SET | ERR_BAUDRATE_INVALID_OR_ALREADY_SET
  102 | DIAG_COMPARE_MISMATCH | DIAG_COMPARE_MISMATCH | DIAG_COMPARE_MISMATCH
  103 | DIAG_COMPARE_MISMATCH_VSYS | DIAG_COMPARE_MISMATCH_VSYS | DIAG_COMPARE_MISMATCH_VSYS
  104 | DIAG_GROUP_OVERLOAD_CURRENT | DIAG_GROUP_OVERLOAD_CURRENT | DIAG_GROUP_OVERLOAD_CURRENT
  105 | ERR_GROUP_OVERLOAD_CURRENT | ERR_GROUP_OVERLOAD_CURRENT | ERR_GROUP_OVERLOAD_CURRENT
  106 | STAT_PAUSED | STAT_PAUSED | STAT_PAUSED
  107 | STAT_ABORT | STAT_ABORT | STAT_ABORT
  108 | STAT_EVNT_OPEN_PLUG_STORAGE | STAT_EVNT_OPEN_PLUG_STORAGE | STAT_EVNT_OPEN_PLUG_STORAGE
  109 | STAT_EVNT_OPEN_UNPLUG_STORAGE | STAT_EVNT_OPEN_UNPLUG_STORAGE | STAT_EVNT_OPEN_UNPLUG_STORAGE
  110 | STAT_EVNT_OPEN_DONE | STAT_EVNT_OPEN_DONE | STAT_EVNT_OPEN_DONE
  111 | STAT_EVNT_REGI_PLUG_STORAGE | STAT_EVNT_REGI_PLUG_STORAGE | STAT_EVNT_REGI_PLUG_STORAGE
  112 | STAT_EVNT_REGI_UNPLUG_STORAGE | STAT_EVNT_REGI_UNPLUG_STORAGE | STAT_EVNT_REGI_UNPLUG_STORAGE
  113 | STAT_EVNT_REGI_DONE | STAT_EVNT_REGI_DONE | STAT_EVNT_REGI_DONE
  114 | STAT_EVNT_UNREGI | STAT_EVNT_UNREGI | STAT_EVNT_UNREGI
  115 | STAT_EVNT_UNREGI_DONE | STAT_EVNT_UNREGI_DONE | STAT_EVNT_UNREGI_DONE
  116 | STAT_EVNT_CLOSE | STAT_EVNT_CLOSE | STAT_EVNT_CLOSE
  117 | STAT_EVNT_CLOSE_DONE | STAT_EVNT_CLOSE_DONE | STAT_EVNT_CLOSE_DONE
  118 | ERR_INSTANCE_RESTRICTION | ERR_INSTANCE_RESTRICTION | ERR_INSTANCE_RESTRICTION
  119 | ERR_NO_FILE | ERR_NO_FILE | ERR_NO_FILE
  120 | ERR_EVNT_OPEN | ERR_EVNT_OPEN | ERR_EVNT_OPEN
  121 | ERR_EVNT_REGI | ERR_EVNT_REGI | ERR_EVNT_REGI
  122 | ERR_EVNT_UNREGI | ERR_EVNT_UNREGI | ERR_EVNT_UNREGI
  123 | ERR_EVNT_CLOSE | ERR_EVNT_CLOSE | ERR_EVNT_CLOSE
  124 | ERR_GET_STORAGE_LIST | ERR_GET_STORAGE_LIST | ERR_GET_STORAGE_LIST
  125 | ERR_UNPLUG_STORAGE | ERR_UNPLUG_STORAGE | ERR_UNPLUG_STORAGE
  126 | DIAG_INVALID_CHANNEL | DIAG_INVALID_CHANNEL | DIAG_INVALID_CHANNEL
  127 | DIAG_INVALID_MODE | DIAG_INVALID_MODE | DIAG_INVALID_MODE
  128 | ERR_H_BRIDGE_TEST | ERR_H_BRIDGE_TEST | ERR_H_BRIDGE_TEST
  129 | ERR_GROUP_SW_TEST | ERR_GROUP_SW_TEST | ERR_GROUP_SW_TEST
  130 | ERR_TX_ERROR | ERR_TX_ERROR | ERR_TX_ERROR
  131 | ERR_RX_ERROR | ERR_RX_ERROR | ERR_RX_ERROR
  132 | DIAG_PHASE_MISSING_B | DIAG_PHASE_MISSING_B | DIAG_PHASE_MISSING_B
  133 | DIAG_PHASE_TOO_MANY_B | DIAG_PHASE_TOO_MANY_B | DIAG_PHASE_TOO_MANY_B
   |  |  |  *)

(* text list TextList_IO_Diag (id | default)
   |  *)

(* text list TL_eKeyMapCodes (id | default)
  0 | NONE
  1 | ESCAPE
  74 | MINUS
  55 | ASTERISK
  57 | SPACE
  83 | COMMA
  98 | SLASH
  78 | PLUS
  11 | KEY_0
  2 | KEY_1
  3 | KEY_2
  4 | KEY_3
  5 | KEY_4
  6 | KEY_5
  7 | KEY_6
  8 | KEY_7
  9 | KEY_8
  10 | KEY_9
  30 | KEY_A
  48 | KEY_B
  46 | KEY_C
  32 | KEY_D
  18 | KEY_E
  33 | KEY_F
  34 | KEY_G
  35 | KEY_H
  23 | KEY_I
  36 | KEY_J
  37 | KEY_K
  38 | KEY_L
  50 | KEY_M
  49 | KEY_N
  24 | KEY_O
  25 | KEY_P
  16 | KEY_Q
  19 | KEY_R
  31 | KEY_S
  20 | KEY_T
  22 | KEY_U
  47 | KEY_V
  17 | KEY_W
  45 | KEY_X
  21 | KEY_Y
  44 | KEY_Z
  28 | KEY_RETURN
  14 | BACKSPACE
  15 | TAB
  99 | PRINT
  102 | HOME
  103 | UP
  105 | LEFT
  106 | RIGHT
  107 | END
  108 | DOWN
  110 | INSERT
  111 | DELETE
  119 | PAUSE
  59 | F1
  60 | F2
  61 | F3
  62 | F4
  63 | F5
  64 | F6
  65 | F7
  66 | F8
  67 | F9
  68 | F10
  87 | F11
  88 | F12
  82 | NUM0
  79 | NUM1
  80 | NUM2
  81 | NUM3
  75 | NUM4
  76 | NUM5
  77 | NUM6
  71 | NUM7
  72 | NUM8
  73 | NUM9
   |  *)
